Staubli VAL3: getLibName.pgx

public program getLibName(string x_slibPath, string& x_sLibName)
begin
  // This program receives the application’s full path, and returns
  //  only the application’s name.
  //
  // Input param
  //  x_slibPath     : Application’s full path
  //
  // Output Param
  //  x_sLibName     : Application’s name
  //
  //----------------------------------------------------------------
  //
  while find(x_slibPath,"/")>-1
    x_slibPath=delete(x_slibPath,find(x_slibPath,"/")+1,0)
  endWhile
  while find(x_slibPath,"\")>-1
    x_slibPath=delete(x_slibPath,find(x_slibPath,"\")+1,0)
  endWhile
  x_sLibName=x_slibPath
end
